PROGRAM MAIN
VAR
END_VAR

END_PROGRAM

(* stored: Version 1.1.0.1, ProductVersion 3.1.0.36
   POU MAIN: Id {95a0d32a-8f7a-417e-8f92-b2750816dffa} *)
